RoboDK station: MCTE4352_1717231.rdk

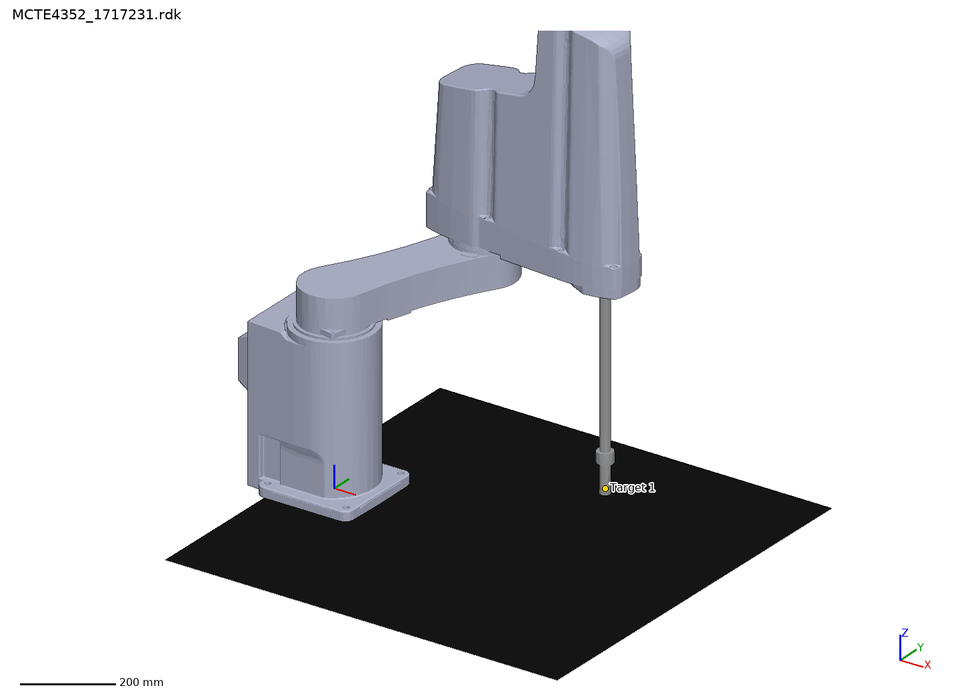
[picture v0: the station drawn from its stored meshes, robots at their saved joint values, targets as dots, program paths as lines]
Station New Station (2) (saved by RoboDK 5.3.3). Poses are relative to the parent item; angles as X-Y-Z fixed-axis rotations.
  - Python program Prog1 (listed below)
  - frame Mitsubishi RH-12FH7035 Base at (-394.52, 0, 0) mm
    - robot Mitsubishi RH-12FH7035: 4 axes, payload 12 kg, reach 600 mm, repeatability 0.025 mm
        modified DH rows (alpha deg, a mm, theta deg, d mm): 0, 0, 0, 0; 0, 375, 0, 0; 0, 325, 0, 0 linear; 180, 0, 0, 0
        joint limits [-132, -150, 0, -360] to [132, 150, 300, 360]; home [0, 0, 350, 0]; saved at [68.005, -72.196, 0, 4.191]
    - target Target 1 (Cartesian target) at (464.58, 323.95, 0) mm; joints [130.825, -126.489, 0, -4.336] of Mitsubishi RH-12FH7035
  - object Plane 1m x 1m at (0, 35.65, -10) mm, size 1000 x 1000 x 0.5 mm, geometry from plane.sld

--- Python program Prog1 ---
# Type help("robolink") or help("robodk") for more information
# Press F5 to run the script
# Documentation: https://robodk.com/doc/en/RoboDK-API.html
# Reference:     https://robodk.com/doc/en/PythonAPI/index.html
# Note: It is not required to keep a copy of this file, your python script is saved with the station

from robolink import *
from robodk import *

path = getOpenFile(r"C:\Users\Hassan Boufares\Downloads\RDK") # Calling the name of the folder to select the .CSV file.
data = LoadList(path) #Loading the names coordinates using LoadList.
RDK = Robolink() #A general referring to the robot that is being used in the project.
robot = RDK.Item('', ITEM_TYPE_ROBOT) #Choosing the robot to apply this program at.
target = RDK.Item('Target 1')
position = target.Pose()
program_name = getFileName(path)
program = RDK.AddProgram(program_name, robot)
RDK.Render(False)

for i in range(len(data)):
    pi = position
    pi.setPos(data[i])
    target.setPose(pi)
    if i == 0:
        robot.MoveJ(target)
    else:

        robot.MoveL(target)

    if i % 100 == 0:
        program.ShowTargets(False)
        RDK.ShowMessage("Loading %s: %.1f %%" % (program, 100*i/len(data)),False)
        RDK.Render()
program.ShowTargets(False)
